FUNCTION_BLOCK NormallyOpenSensor
VAR
	input AT %I*	:	BOOL;
END_VAR

PROPERTY PUBLIC IsActive : BOOL

// ho eliminato manualmente il Setter di questa proprietà perché qui non ha senso
GET
IsActive := input;
END_GET
END_PROPERTY

END_FUNCTION_BLOCK

(* stored: Version 1.1.0.1, ProductVersion 3.1.4024.11
   POU NormallyOpenSensor: Id {b620ad30-adc5-4dbe-82d7-016f9c37814d}, SpecialFunc None
   Property IsActive: Id {7804bb6d-2964-4334-af99-f7c637281512}
   Get Get: Id {c46e44ec-8482-459a-a039-a63f5f84f4cd} *)
